SUBAPPLICATION mapping_Uebung_060 (* für TC-SC also Task Controller Section Control *)
  (* Standard: 61499-2; Description: Copyright (c) 2023 Meisterschulen am Ostbahnhof This program and the accompanying materials are made available under the terms of the Eclipse Public License 2.0 which is available at https://www.eclipse.org/legal/epl-2.0/ SPDX-License-Identifier: EPL-2.0 *)
  (* Version 1.0, 2023-10-23, Franz Höpfinger, Meisterschulen am Ostbahnhof *)
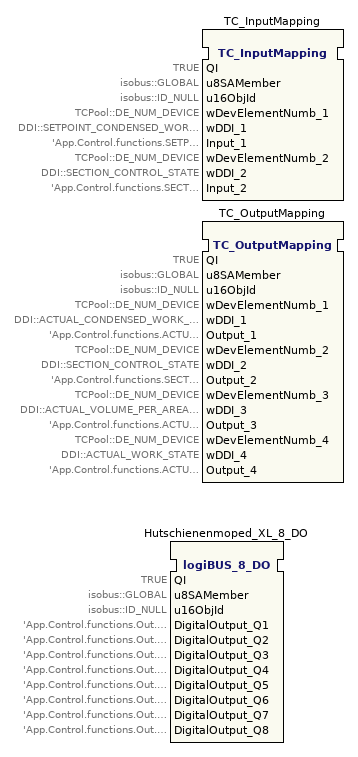
  FBS
    TC_InputMapping : TC_InputMapping(QI := TRUE, u8SAMember := isobus::GLOBAL, u16ObjId := isobus::ID_NULL, wDevElementNumb_1 := TCPool::DE_NUM_DEVICE, wDDI_1 := DDI::SETPOINT_CONDENSED_WORK_STATE_1_16, Input_1 := 'App.Control.functions.SETPOINT_CONDENSED_WORK_STATE_1_16', wDevElementNumb_2 := TCPool::DE_NUM_DEVICE, wDDI_2 := DDI::SECTION_CONTROL_STATE, Input_2 := 'App.Control.functions.SECTION_CONTROL_STATE_IN');
    TC_OutputMapping : TC_OutputMapping(QI := TRUE, u8SAMember := isobus::GLOBAL, u16ObjId := isobus::ID_NULL, wDevElementNumb_1 := TCPool::DE_NUM_DEVICE, wDDI_1 := DDI::ACTUAL_CONDENSED_WORK_STATE_1_16, Output_1 := 'App.Control.functions.ACTUAL_CONDENSED_WORK_STATE_1_16', wDevElementNumb_2 := TCPool::DE_NUM_DEVICE, wDDI_2 := DDI::SECTION_CONTROL_STATE, Output_2 := 'App.Control.functions.SECTION_CONTROL_STATE_OUT', wDevElementNumb_3 := TCPool::DE_NUM_DEVICE, wDDI_3 := DDI::ACTUAL_VOLUME_PER_AREA_APPLICATION_RATE, Output_3 := 'App.Control.functions.ACTUAL_RATE', wDevElementNumb_4 := TCPool::DE_NUM_DEVICE, wDDI_4 := DDI::ACTUAL_WORK_STATE, Output_4 := 'App.Control.functions.ACTUAL_WORK_STATE');
    Hutschienenmoped_XL_8_DO : logiBUS_8_DO(QI := TRUE, u8SAMember := isobus::GLOBAL, u16ObjId := isobus::ID_NULL, DigitalOutput_Q1 := 'App.Control.functions.Out.DigitalOutput_Q1', DigitalOutput_Q2 := 'App.Control.functions.Out.DigitalOutput_Q2', DigitalOutput_Q3 := 'App.Control.functions.Out.DigitalOutput_Q3', DigitalOutput_Q4 := 'App.Control.functions.Out.DigitalOutput_Q4', DigitalOutput_Q5 := 'App.Control.functions.Out.DigitalOutput_Q5', DigitalOutput_Q6 := 'App.Control.functions.Out.DigitalOutput_Q6', DigitalOutput_Q7 := 'App.Control.functions.Out.DigitalOutput_Q7', DigitalOutput_Q8 := 'App.Control.functions.Out.DigitalOutput_Q8');
  END_FBS
END_SUBAPPLICATION
